// TIA Portal V19 export
DATA_BLOCK "DataFromStandard"   // DB128
// stored: InstanceOfName Safety.typeDataToSafety, InstanceOfType UDT, Namespace Safety
"Safety.typeDataToSafety"
   // VAR
   //    ackSafetyFromHmi : Int;
   //    ackSafetyGlobal : Bool;
   //    ackFromUnit : Bool;
   // END_VAR
BEGIN
END_DATA_BLOCK
